TYPE Heating_Ctx_Io :
STRUCT
	in		: Heating_Ctx_Io_In;
	out		: Heating_Ctx_Io_Out;
END_STRUCT
END_TYPE

(* stored: Version 1.1.0.1
   DUT Heating_Ctx_Io: Id {ab002f6c-aa25-453a-80cc-9323ae49b2c1} *)
